FUNCTION_BLOCK FB_BaseControlElement_HMI EXTENDS FB_BaseComponent_HMI IMPLEMENTS ITF_BaseControlElement_HMI
VAR
	itfBaseControlElementConnector		: ITF_BaseControlElement_HMI_Connector;
	refstBaseControlElementDataHMI		: REFERENCE TO ST_BaseControlElement_HMI;
	(*	lista componentów składających się na ten element w elemencie docelowym dodać itf dla konkretnych elementów	*)
	arrComponent						: ARRAY  [1..GVL_BaseConstans.MAX_ITEM_PER_ELEMENT] OF ITF_BaseComponent_HMI;
	uiNumberOfComponents				: UINT;

END_VAR

METHOD PROTECTED AddComponent : BOOL
VAR_INPUT
	itfComponentHMI				: ITF_BaseComponent_HMI;
END_VAR
IF (THIS^.uiNumberOfComponents + 1 <= GVL_BaseConstans.MAX_ITEM_PER_ELEMENT) THEN
	THIS^.uiNumberOfComponents		:= THIS^.uiNumberOfComponents + 1;
	THIS^.arrComponent [THIS^.uiNumberOfComponents]	:= itfComponentHMI;
	AddComponent				:= TRUE;
ELSE
	;//zwrocenie zbyt dużo komponentow
END_IF
END_METHOD

END_FUNCTION_BLOCK

(* stored: Version 1.1.0.1
   POU FB_BaseControlElement_HMI: Id {f7e14e4d-7841-0cfb-1cf8-aac3b29affb7}, SpecialFunc None
   Method AddComponent: Id {d792cffc-9654-05bf-1253-a43b4835c74a} *)
